// TIA Portal V20 export
DATA_BLOCK "HmiInterface"   // DB68
// stored: Access Published, MemoryReserve 100, Namespace Unit1.Em7
   VAR
      em : "LAF_typeEmInterface";
      hotPressRight : "LER_typeSequenceInterface";
      cmHotPressRightSafetyPin : "LBC_typeDigitalSignalInterface";
      cmHotPressRightJRDetect : "LBC_typeDigitalSignalInterface";
      cmHotPressRightStageLiftFrontUpDown : "LBC_typeTwoWayActuatorInterface";
      cmHotPressRightStageLiftRearUpDown : "LBC_typeTwoWayActuatorInterface";
      cmHotPressRightStageLiftAllUpDown : "LBC_typeTwoWayActuatorInterface";
      cmHotPressRightServoPress : "LER_typeServoPressInterface";
      cmHotPressRightTemperature : "LER_typeHeaterInterface";
   END_VAR
   VAR RETAIN
      cmHotPressRightHistory : "LER_typeServoPressHistory";
   END_VAR
   VAR
      intCondition : "Unit1.Em7.typeIntConditionHmiInterface";
   END_VAR
BEGIN
   cmHotPressRightTemperature.configuration.E5CC[1..5].Temp_SP := 0;
   cmHotPressRightTemperature.configuration.E5CC[1..5].Temp_AlarmValue1 := 0;
   cmHotPressRightTemperature.configuration.E5CC[1..5].Temp_AlarmValue1_UpperLimit := 45;
   cmHotPressRightTemperature.configuration.E5CC[1..5].Temp_AlarmValue1_LowerLimit := 15;
   cmHotPressRightTemperature.configuration.E5CC[1..5].Temp_AlarmValue2 := 0;
   cmHotPressRightTemperature.configuration.E5CC[1..5].Temp_AlarmValue2_UpperLimit := 42;
   cmHotPressRightTemperature.configuration.E5CC[1..5].Temp_AlarmValue2_LowerLimit := 18;
   cmHotPressRightTemperature.configuration.E5CC[1..5].Temp_Upper_Limit_Temp := 40;
   cmHotPressRightTemperature.configuration.E5CC[1..5].Temp_Lower_Limit_Temp := 20;
   cmHotPressRightTemperature.configuration.E5CC[1..5].Temp_MC_Off_Value := 0;
   cmHotPressRightTemperature.configuration.E5CC[1..5].Temp_Upper_Complete_Range := 1;
   cmHotPressRightTemperature.configuration.E5CC[1..5].Temp_Lower_Complete_Range := -1;
END_DATA_BLOCK
